// TIA Portal V19 export
DATA_BLOCK "A0303_Spalla_Pers"   // DB93
// stored: MemoryReserve 100
   VAR RETAIN
      Par : Struct
         Testa : Struct
            Ax : "Positioning_DOL_Machine_Par";
            Ax_Pers : "Positioning_DOL_Machine_Pers_Data";
            Enc : "PosFbk_RTN";
         END_STRUCT;
         Coda : Struct
            Ax : "Positioning_DOL_Machine_Par";
            Ax_Pers : "Positioning_DOL_Machine_Pers_Data";
            Enc : "PosFbk_RTN";
         END_STRUCT;
      END_STRUCT;
      Par_Mach_Testa : Struct
         MinDistanzaConParegg { S7_SetPoint := 'True'} : LReal := -10.0;
         ToleranceWindow : LReal := 0.5;
      END_STRUCT;
      Par_Mach_Coda : Struct
         MinDistanzaConParegg : LReal := -100.0;
         ToleranceWindow : LReal := 0.2;
      END_STRUCT;
   END_VAR
BEGIN
   Par.Testa.Ax.PosTolerance := 0.5;
   Par.Testa.Ax.Minus_Limit := 83.0;
   Par.Testa.Ax.Plus_Limit := 2730.0;
   Par.Testa.Ax.PreCutOff := 0.0;
   Par.Testa.Ax.PreEndLowSpeed := 5.0;
   Par.Testa.Ax.PreEndMedSpeed := 10.0;
   Par.Testa.Ax.LowSpeed := 2.0;
   Par.Testa.Ax.MedSpeed := 10.0;
   Par.Testa.Ax.HighSpeed := 50.0;
   Par.Testa.Ax.Man_Speed := 50.0;
   Par.Testa.Ax_Pers.AxisHomed := TRUE;
   Par.Testa.Enc.Preset.Pulses := 2_098_215_900;
   Par.Testa.Enc.Preset.Units := 913.0;
   Par.Testa.Enc.Config.Resolution := 376.9911168;
   Par.Coda.Ax.PosTolerance := 0.5;
   Par.Coda.Ax.Minus_Limit := 80.0;
   Par.Coda.Ax.Plus_Limit := 2730.0;
   Par.Coda.Ax.PreCutOff := 0.2;
   Par.Coda.Ax.PreEndLowSpeed := 2.0;
   Par.Coda.Ax.PreEndMedSpeed := 5.0;
   Par.Coda.Ax.LowSpeed := 5.0;
   Par.Coda.Ax.MedSpeed := 10.0;
   Par.Coda.Ax.HighSpeed := 50.0;
   Par.Coda.Ax.Man_Speed := 50.0;
   Par.Coda.Ax_Pers.AxisHomed := TRUE;
   Par.Coda.Enc.Preset.Pulses := 14325816;
   Par.Coda.Enc.Preset.Units := 913.0;
   Par.Coda.Enc.Config.Resolution := -376.9911168;
END_DATA_BLOCK
